// TIA Portal V16 export
// export: Created 2021-05-26T11:52:20.8559157Z, ExportSetting WithDefaults, DisplayName Totally Integrated Automation Portal, DisplayVersion V16 Update 4, DisplayName TIA Portal Version Control Interface, DisplayVersion V16 Update 2, DisplayName TIA Portal Openness, DisplayVersion V16 Update 4, DisplayName STEP 7 Professional, DisplayVersion V16 Update 4, DisplayName STEP 7 Safety, DisplayVersion V16, DisplayName WinCC Advanced, DisplayVersion V16 Update 4
DATA_BLOCK "DB_DrvCon"   // DB36
{ S7_Optimized_Access := 'FALSE' }
VERSION : 0.1
// stored: AutoNumber true, DBAccessibleFromOPCUA true, IsOnlyStoredInLoadMemory false, IsWriteProtectedInAS false
   VAR
      Data_Send : Struct
         SwpStartTime : Int;
         SwpTimeStep : Int;
         sweepMod : Byte;
         stOFF : Bool;
         res_b5_bit1 : Bool;
         res_b5_bit2 : Bool;
         res_b5_bit3 : Bool;
         res_b5_bit4 : Bool;
         res_b5_bit5 : Bool;
         res_b5_bit6 : Bool;
         res_b5_bit7 : Bool;
         CommCnt : Byte;
      END_STRUCT;
      Data_Rcv : Struct
         CurDrvTr1 : Int;
         CurDrvTr2 : Int;
         CurDrvTr3 : Int;
         CurDrvTr4 : Int;
         CurDrvTr5 : Int;
         CurDrvTr6 : Int;
         CurDrvTr7 : Int;
         CurDrvTr8 : Int;
         CurDrvTr9 : Int;
         CurDrvTr10 : Int;
         CurDrvTr11 : Int;
         CurDrvTr12 : Int;
         CurDrvTr13 : Int;
         CurDrvTr14 : Int;
         CurDrvTr15 : Int;
         CurDrvTr16 : Int;
         CurPrDrv2Stg2 : Int;
         CurPrDrv2Stg3 : Int;
         spare1 : Int;
         spare2 : Int;
         spare3 : Int;
         spare4 : Int;
         spare5 : Int;
         spare6 : Int;
         VoltDrvTr1 : Int;
         VoltDrvTr2 : Int;
         VoltDrvTr3 : Int;
         VoltDrvTr4 : Int;
         VoltDrvTr5 : Int;
         VoltDrvTr6 : Int;
         VoltDrvTr7 : Int;
         VoltDrvTr8 : Int;
         VoltDrvTr9 : Int;
         VoltDrvTr10 : Int;
         VoltDrvTr11 : Int;
         VoltDrvTr12 : Int;
         VoltDrvTr13 : Int;
         VoltDrvTr14 : Int;
         VoltDrvTr15 : Int;
         VoltDrvTr16 : Int;
         VoltPDrv2Stg2 : Int;
         VoltPDrv2Stg3 : Int;
         spare7 : Int;
         spare8 : Int;
         spare9 : Int;
         spare10 : Int;
         spare11 : Int;
         spare12 : Int;
         TmpMB1_Drv : Int;
         TmpMB2 : Int;
         TmpMB3_PrD : Int;
         DrvDataTr : Array[1..8] of "UDT_swp51Data";
         sweepIV { S7_SetPoint := 'True'} : Bool;
         stTrigger { S7_SetPoint := 'True'} : Bool;
         ModConnect1 { S7_SetPoint := 'True'} : Bool;
         ModConnect2 : Bool;
         ModTmpSw1 : Bool;
         ModTmpSw2 : Bool;
         res_b882_6 : Bool;
         res_b882_7 : Bool;
         sweepMB : Byte;
         SoftVersion : Byte;
         CommCntRB : Byte;
      END_STRUCT;
   END_VAR
BEGIN
END_DATA_BLOCK
